Staubli VAL3: SA.pgx

public program SA(dio x_dInput, dio x_dOutput, num x_nLength)
begin

  //"reset delay"
  //reset the x_dOutput only when x_dInput is false for a time greater than x_nLength
  //note: x_dInput isn't necessarily an input

  if taskStatus("SA_"+toString("",nSA_Count))==-1
    taskCreate "SA_"+toString("",nSA_Count),10,exeSA(x_dInput,x_dOutput,x_nLength)
    nSA_Count=nSA_Count+1
    if nSA_Count>nMaxTask
      nSA_Count=0
    endIf
  else
    logMsg("libSignals/SA->can't create SA task")
  endIf

end
